ABB RobotStudio station: PicknPlace.rspag

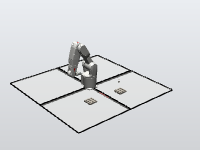
--- station ---
Station PickUp Test_3 (saved by RobotStudio 6.8.8148.134)
Controller IRB_1200_5kg_0.9m
  mechanical unit ROB_1: IRB1200FPL_5_90_STD_01, 6 joints, base frame (0, 0, 0) mm
Layout (positions relative to the parent item):
  - IRB1200FPL_5_90_STD_01 [mechanism, from Robots\IRB1200FPL_5_90_STD_01.rslib] at (0, 0, 0) mm; joint values [-1.5708, 0.5236, 0.7854, 0, 1.5708, -1.5708] (rad or m)
  - Smart_Gripper_Servo_Fingers [mechanism, from Tools\ABB_Smart_Gripper_Servo_Fingers.rslib] at (0, -302.09, 341.1) mm, rotated rx 105 ry 0 rz 180 deg; joint values [0.02] (rad or m)
  - Peg [part] at (200, 500, 0) mm
  - Plate_A [part] at (400, 200, 0) mm
  - Plate_B [part] at (350, -400, 0) mm
  - LineSensor [smart component, from Components\LineSensor.rslib] at (0, -196.61, 312.83) mm, rotated rx 105 ry 0 rz 180 deg
      properties: Start=[0.0200323016476803 -1.83356878054597E-05 0.0210805401622316]; End=[-0.0201221711320567 1.77313040473637E-05 0.021186539942684]; Radius=0.005; SensedPart=(none); SensedPoint=[0 0 0]
    - _sensorPart_ [part]
  - Attacher [smart component, from Components\Attacher.rslib]
      properties: Parent=IRB1200FPL_5_90_STD_01; Flange=0; Child=(none); Mount=false; Offset=[0 0 0]; Orientation=[0 0 0]
  - Detacher [smart component, from Components\Detacher.rslib]
      properties: Child=(none); KeepPosition=true
  - PoseMover [smart component, from Components\PoseMover.rslib]
      properties: Mechanism=Smart_Gripper_Servo_Fingers; Pose=2; Duration=0
  - PoseMover_2 [smart component, from Components\PoseMover.rslib]
      properties: Mechanism=Smart_Gripper_Servo_Fingers; Pose=3; Duration=0
Attachment: Smart_Gripper_Servo_Fingers is attached to IRB1200FPL_5_90_STD_01 / Link6
Attachment: LineSensor is attached to Smart_Gripper_Servo_Fingers / HandBase
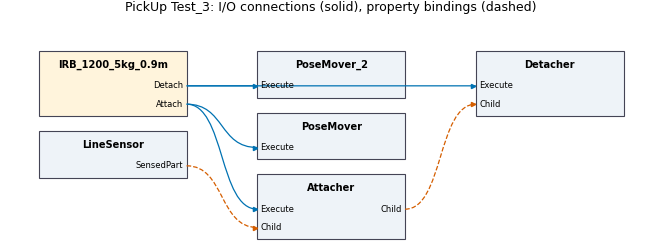
Station logic (signal -> signal, property => property):
  IRB_1200_5kg_0.9m.Detach -> Detacher.Execute
  IRB_1200_5kg_0.9m.Attach -> Attacher.Execute
  IRB_1200_5kg_0.9m.Detach -> PoseMover_2.Execute
  IRB_1200_5kg_0.9m.Attach -> PoseMover.Execute
  Attacher.Child => Detacher.Child
  LineSensor.SensedPart => Attacher.Child
Targets, tools, work objects and paths stored in the station and not in the controller backup, written as RAPID:
! task T_ROB1
MODULE BASE
  PERS wobjdata wobj_gripper:=[FALSE,TRUE,"",[[0,0,0],[1,0,0,0]],[[0,0,0],[1,0,0,0]]];
ENDMODULE


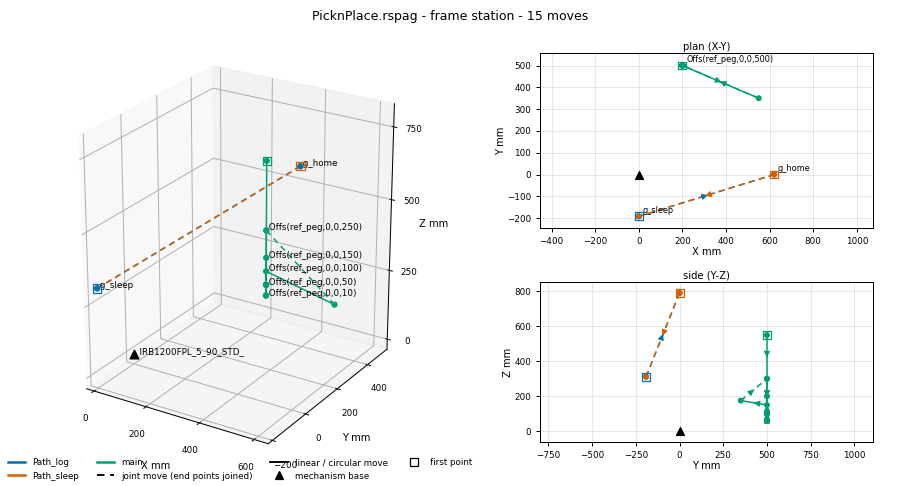
[picture p0: tool path of PicknPlace.rspag in frame station, 15 of 26 moves have a stored position in this frame; points joined in program order, loops and branches not executed]
--- Backups/IRB_1200_5kg_0.9m/RAPID/TASK1/PROGMOD/Module1.mod ---
MODULE Module1

    CONST robtarget g_sleep:=[[0.0,-191.78,311.54],[0,0,0.79335,0.60876],[-1,0,-1,0],[9E+09,9E+09,9E+09,9E+09,9E+09,9E+09]];
    CONST robtarget g_home:=[[620.91,0.0,791.0],[0.35355,-0.61237,0.61237,-0.35355],[0,0,-1,0],[9E+09,9E+09,9E+09,9E+09,9E+09,9E+09]];
    CONST robtarget ref_peg:=[[200,500,50],[0,0.923879533,-0.382683432,0],[0,0,0,0],[9E+09,9E+09,9E+09,9E+09,9E+09,9E+09]];
    CONST robtarget ref_plateA:=[[550,350,25],[0,-0.707106781,0.707106781,0],[0,0,0,0],[9E+09,9E+09,9E+09,9E+09,9E+09,9E+09]];
    CONST robtarget ref_plateB:=[[400,-250,25],[0,-0.707106781,0.707106781,0],[0,0,0,0],[9E+09,9E+09,9E+09,9E+09,9E+09,9E+09]];
    CONST robtarget f_plateA:=[[525,325,25],[0,0.866025404,-0.5,0],[0,0,0,0],[9E+09,9E+09,9E+09,9E+09,9E+09,9E+09]];
    CONST robtarget f_plateB:=[[475.000398044,-275.000229832,25],[0,-0.5,0.866025404,0],[-1,0,-2,0],[9E+09,9E+09,9E+09,9E+09,9E+09,9E+09]];

    CONST num SafetyZ_Offset:=150;
    CONST num Xinc:=-50;
    CONST num Yinc:=-50;
    VAR num Xpos:=0;
    VAR num Ypos:=0;
    PERS tooldata Gripper:=[TRUE,[[0,0,114.2],[1,0,0,0]],[0.215,[8.7,12.3,49.2],[1,0,0,0],0.00021,0.00024,0.00009]];

    PROC Path_log()
        MoveJ g_sleep,v400,z10,Gripper\WObj:=wobj0;
        MoveJ g_home,v600,z10,Gripper\WObj:=wobj0;
    ENDPROC

    PROC Path_sleep()
        MoveJ g_home,v600,z10,Gripper\WObj:=wobj0;
        MoveJ g_sleep,v400,z10,Gripper\WObj:=wobj0;
    ENDPROC

    PROC DoAttach()
        SetDO Attach,1;
        WaitTime 0.35;
        SetDO Attach,0;
        WaitTime 0.15;
    ENDPROC

    PROC DoDetach()
        SetDO Detach,1;
        WaitTime 0.35;
        SetDO Detach,0;
        WaitTime 0.15;
    ENDPROC

    PROC PicknPlace()
        MoveJ Offs(f_plateA,Xpos,Ypos,SafetyZ_Offset),v800,fine,Gripper\WObj:=wobj0;
        MoveL Offs(f_plateA,Xpos,Ypos,100),v600,fine,Gripper\WObj:=wobj0;
        MoveL Offs(f_plateA,Xpos,Ypos,50),v500,fine,Gripper\WObj:=wobj0;
        DoDetach;
        MoveL Offs(f_plateA,Xpos,Ypos,100),v800,fine,Gripper\WObj:=wobj0;
        MoveL Offs(f_plateA,Xpos,Ypos,50),v500,fine,Gripper\WObj:=wobj0;
        DoAttach;
        MoveL Offs(f_plateA,Xpos,Ypos,SafetyZ_Offset),v800,fine,Gripper\WObj:=wobj0;
        MoveL Offs(f_plateB,Xpos,Ypos,SafetyZ_Offset),v600,fine,Gripper\WObj:=wobj0;
        MoveL Offs(f_plateB,Xpos,Ypos,50),v500,fine,Gripper\WObj:=wobj0;
        DoDetach;
        MoveL Offs(f_plateB,Xpos,Ypos,SafetyZ_Offset),v800,fine,Gripper\WObj:=wobj0;
        MoveL Offs(f_plateB,Xpos,Ypos,50),v500,fine,Gripper\WObj:=wobj0;
        DoAttach;
        MoveL Offs(f_plateB,Xpos,Ypos,SafetyZ_Offset),v600,fine,Gripper\WObj:=wobj0;
    ENDPROC


    PROC main()
        Path_log;
        MoveJ Offs(ref_peg,0,0,500),v500,z50,Gripper\WObj:=wobj0;
        MoveL Offs(ref_peg,0,0,250),v400,z30,Gripper\WObj:=wobj0;
        MoveL Offs(ref_peg,0,0,50),v300,z10,Gripper\WObj:=wobj0;
        MoveL Offs(ref_peg,0,0,10),v200,fine,Gripper\WObj:=wobj0;
        DoAttach;
        MoveL Offs(ref_peg,0,0,100),v500,z20,Gripper\WObj:=wobj0;
        MoveL Offs(ref_plateA,0,0,150),v500,z10,Gripper\WObj:=wobj0;

        FOR Y FROM 0 TO 2 DO
            FOR X FROM 0 TO 2 DO
                PicknPlace;
                Xpos:=Xpos+Xinc;
            ENDFOR
            Ypos:=Ypos+Yinc;
            Xpos:=0;
        ENDFOR
        Ypos:=0;
        MoveJ Offs(ref_peg,0,0,250),v800,z30,Gripper\WObj:=wobj0;
        MoveL Offs(ref_peg,0,0,50),v500,z10,Gripper\WObj:=wobj0;
        MoveL Offs(ref_peg,0,0,10),v200,fine,Gripper\WObj:=wobj0;
        DoDetach;
        MoveL Offs(ref_peg,0,0,50),v500,z10,Gripper\WObj:=wobj0;
        MoveL Offs(ref_peg,0,0,150),v800,z30,Gripper\WObj:=wobj0;
        Path_sleep;
    ENDPROC
ENDMODULE

--- Backups/IRB_1200_5kg_0.9m/SYSPAR/EIO.cfg ---
EIO:CFG_1.0:6:1::
#
EIO_SIGNAL:

      -Name "Attach" -SignalType "DO"

      -Name "Detach" -SignalType "DO"
